FUNCTION TFWorkflowsCheckState : BOOL
VAR_INPUT
	WorkFlow : POINTER TO ARRAY[0..MAXWORKFLOW] OF WorkFlow;
	State : UINT; // stato da verificare
END_VAR
VAR
	i: UINT;
END_VAR
//Funzione che restituisce TRUE se tutti i WORFLOW sono nello stato richiesto

FOR i:=0 TO MAXWORKFLOW DO
	IF WorkFlow^[i].State <> State THEN
		RETURN;
	END_IF
END_FOR
TFWorkflowsCheckState := TRUE;

END_FUNCTION

(* stored: Version 1.1.0.1, ProductVersion 3.1.4024.11
   POU TFWorkflowsCheckState: Id {2a634cf7-cf13-4d64-8bbb-4ed28548e526}, SpecialFunc None *)
